(* Schneider Machine Expert - Basic project Water_Heater, file version 1.8.0.0 *)
(* ProjectInformations: Name=New project *)

HARDWARE
  Cpu 0: TM221ME16T/G
  EthernetConfiguration: NetworkName=M221, IpAllocationMode=FixedAddress, IpAddress=100.100.100.102, SubnetMask=255.0.0.0
  SerialLineConfiguration: Baud=Baud19200, Parity=ParityEven, DataBits=DataBits8, StopBits=StopBits1, PhysicalMedium=PhysicalMediumRs485, TransmissionMode=TransmissionModeModbusRtu, SlaveId=1, Addressing=SlaveAddressing
  MastTask: UsePeriodScanMode=false, PeriodScan=100
  FastTask: Period=255
  CpuBehavior: StartingMode=StartAsPreviousState, AutoSaveRamOnEeprom=true, WatchdogPeriod=250

SYMBOLS  (address, symbol, comment, settings)
  %M0       HEATER_MIRROR
  %M1       HEATER_AUTO
  %M2       HEATER_MAN
  %S13      SB_FIRSTRUN  "Indicates the first controller cycle in RUN mode"
  %MW1      CONVERTED_TEMP
  %MW2      SETPOINT
  %MW3      SETPOINT_MIN
  %MW4      MODE_REGISTER
  %MW5      HEATER_CONTROL
  %Q0.0     HEATER

POU New POU
  (* SectionNumber=1 *)

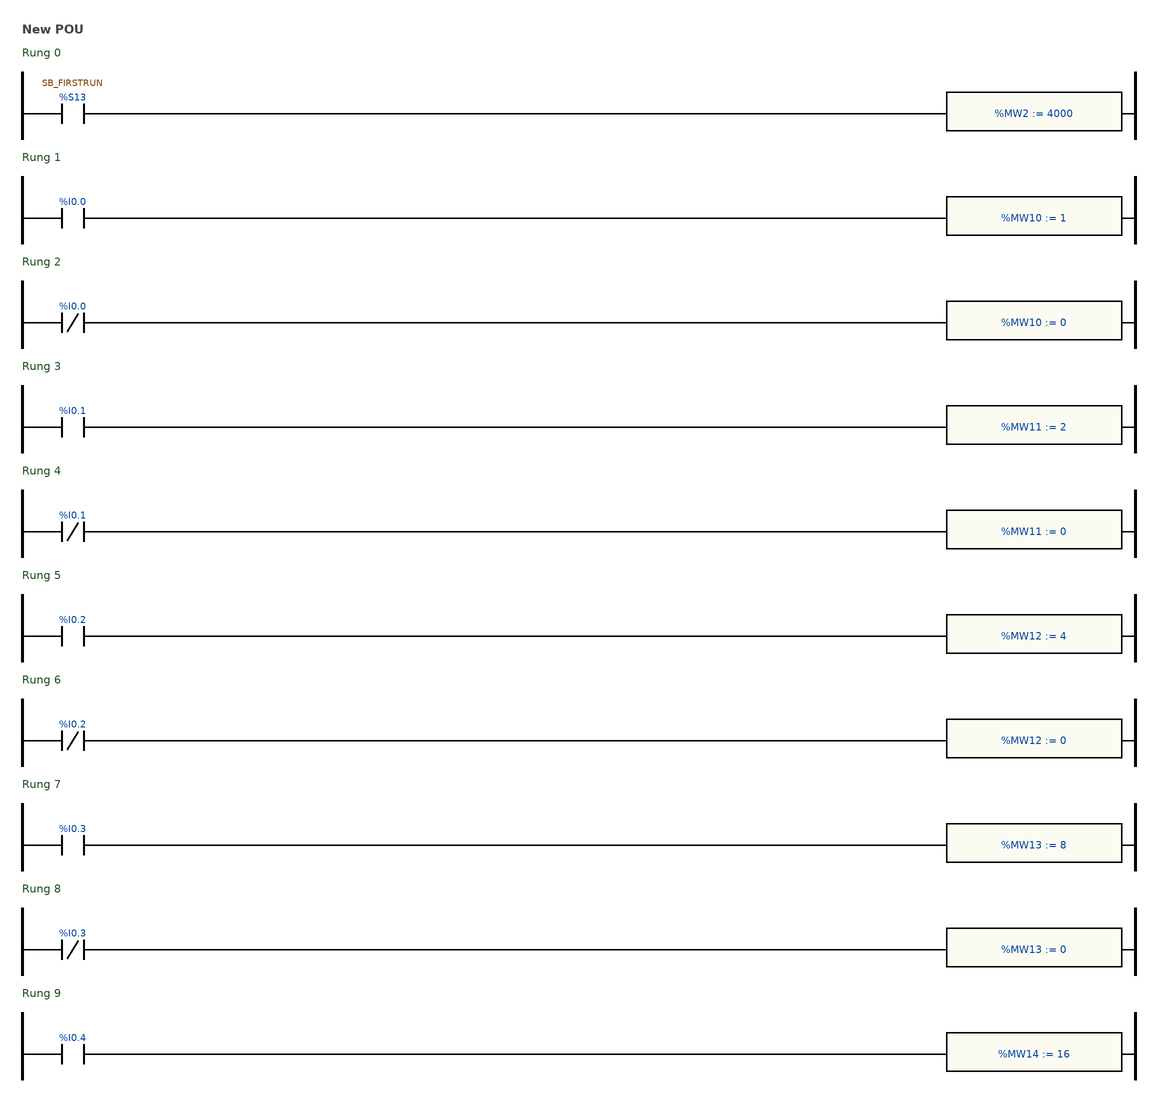

// Rung 0
  LD %S13                 (* SB_FIRSTRUN *)
  [ %MW2 := 4000 ]        (* SETPOINT *)
  // as ST:
  //   IF SB_FIRSTRUN THEN SETPOINT := 4000; END_IF;

// Rung 1
  LD %I0.0
  [ %MW10 := 1 ]
  // as ST:
  //   IF %I0.0 THEN %MW10 := 1; END_IF;

// Rung 2
  LDN %I0.0
  [ %MW10 := 0 ]
  // as ST:
  //   IF NOT %I0.0 THEN %MW10 := 0; END_IF;

// Rung 3
  LD %I0.1
  [ %MW11 := 2 ]
  // as ST:
  //   IF %I0.1 THEN %MW11 := 2; END_IF;

// Rung 4
  LDN %I0.1
  [ %MW11 := 0 ]
  // as ST:
  //   IF NOT %I0.1 THEN %MW11 := 0; END_IF;

// Rung 5
  LD %I0.2
  [ %MW12 := 4 ]
  // as ST:
  //   IF %I0.2 THEN %MW12 := 4; END_IF;

// Rung 6
  LDN %I0.2
  [ %MW12 := 0 ]
  // as ST:
  //   IF NOT %I0.2 THEN %MW12 := 0; END_IF;

// Rung 7
  LD %I0.3
  [ %MW13 := 8 ]
  // as ST:
  //   IF %I0.3 THEN %MW13 := 8; END_IF;

// Rung 8
  LDN %I0.3
  [ %MW13 := 0 ]
  // as ST:
  //   IF NOT %I0.3 THEN %MW13 := 0; END_IF;

// Rung 9
  LD %I0.4
  [ %MW14 := 16 ]
  // as ST:
  //   IF %I0.4 THEN %MW14 := 16; END_IF;

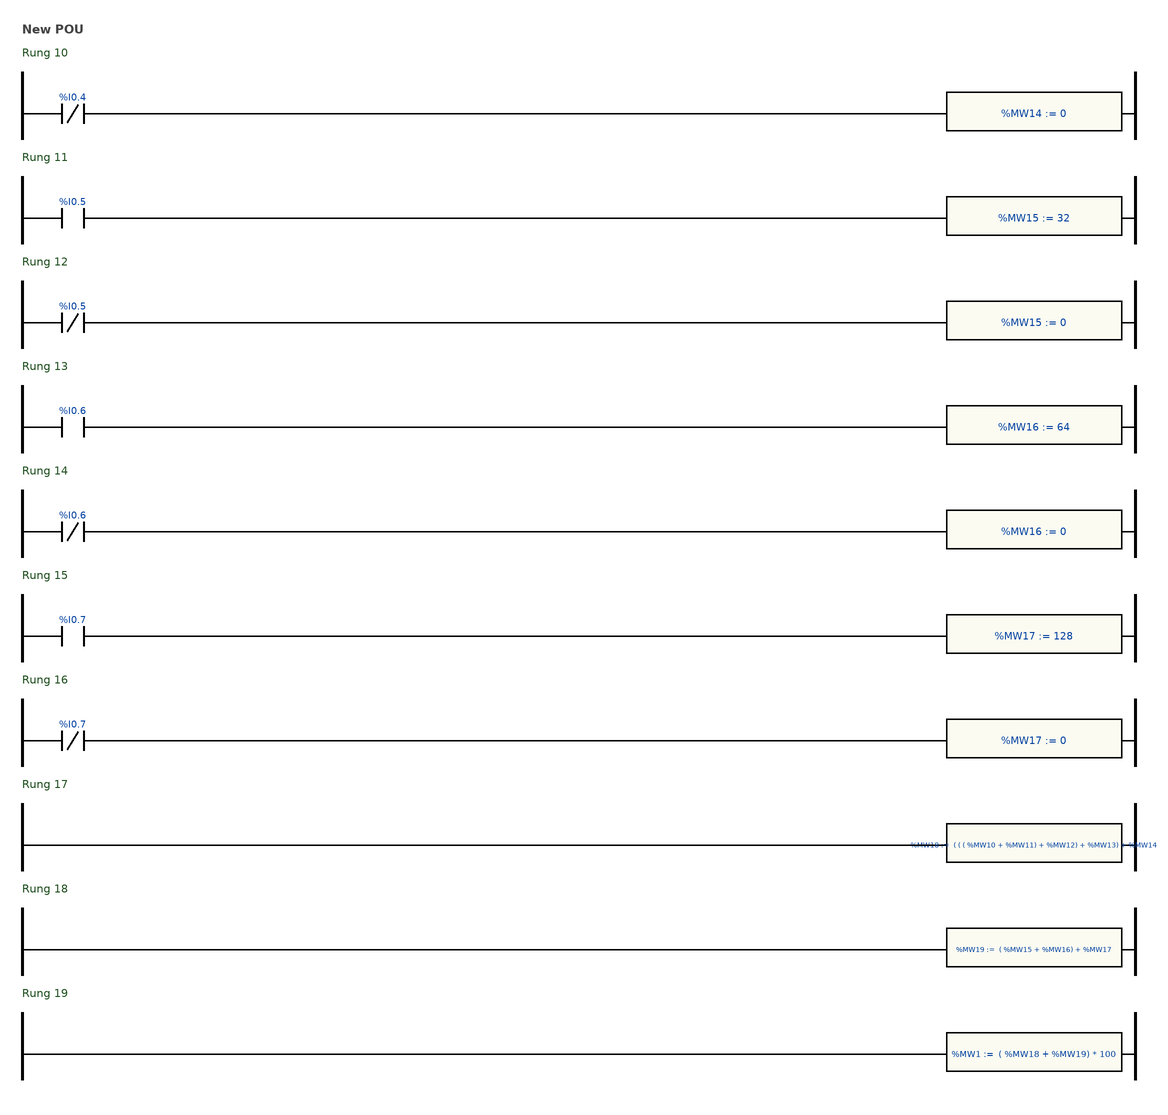

// Rung 10
  LDN %I0.4
  [ %MW14 := 0 ]
  // as ST:
  //   IF NOT %I0.4 THEN %MW14 := 0; END_IF;

// Rung 11
  LD %I0.5
  [ %MW15 := 32 ]
  // as ST:
  //   IF %I0.5 THEN %MW15 := 32; END_IF;

// Rung 12
  LDN %I0.5
  [ %MW15 := 0 ]
  // as ST:
  //   IF NOT %I0.5 THEN %MW15 := 0; END_IF;

// Rung 13
  LD %I0.6
  [ %MW16 := 64 ]
  // as ST:
  //   IF %I0.6 THEN %MW16 := 64; END_IF;

// Rung 14
  LDN %I0.6
  [ %MW16 := 0 ]
  // as ST:
  //   IF NOT %I0.6 THEN %MW16 := 0; END_IF;

// Rung 15
  LD %I0.7
  [ %MW17 := 128 ]
  // as ST:
  //   IF %I0.7 THEN %MW17 := 128; END_IF;

// Rung 16
  LDN %I0.7
  [ %MW17 := 0 ]
  // as ST:
  //   IF NOT %I0.7 THEN %MW17 := 0; END_IF;

// Rung 17
  LD 1
  [%MW18 := ( ( ( %MW10 + %MW11) + %MW12) + %MW13) + %MW14]
  // as ST:
  //   %MW18 :=  ( ( ( %MW10 + %MW11) + %MW12) + %MW13) + %MW14;

// Rung 18
  LD 1
  [%MW19 := ( %MW15 + %MW16) + %MW17]
  // as ST:
  //   %MW19 :=  ( %MW15 + %MW16) + %MW17;

// Rung 19
  LD 1
  [%MW1 := ( %MW18 + %MW19) * 100](* CONVERTED_TEMP *)
  // as ST:
  //   CONVERTED_TEMP :=  ( %MW18 + %MW19) * 100;

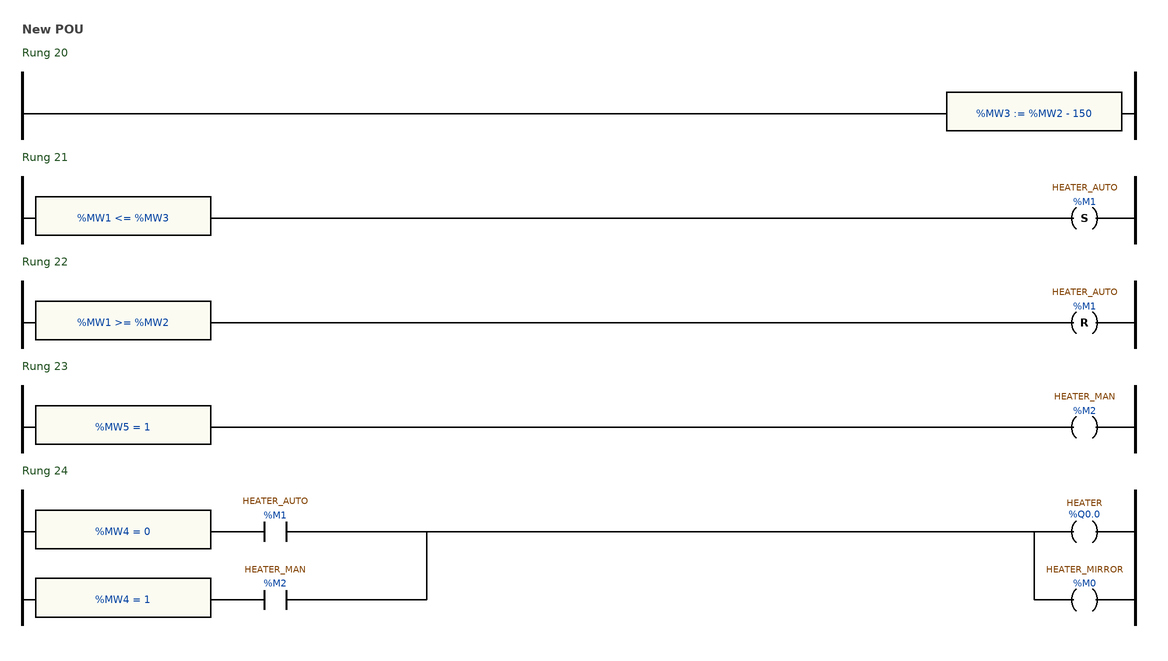

// Rung 20
  LD 1
  [ %MW3 := %MW2 - 150 ]  (* SETPOINT_MIN, SETPOINT *)
  // as ST:
  //   SETPOINT_MIN := SETPOINT - 150;

// Rung 21
  LD [ %MW1 <= %MW3 ]     (* CONVERTED_TEMP, SETPOINT_MIN *)
  S %M1                   (* HEATER_AUTO *)
  // as ST:
  //   IF CONVERTED_TEMP <= SETPOINT_MIN THEN HEATER_AUTO := TRUE; END_IF;

// Rung 22
  LD [ %MW1 >= %MW2 ]     (* CONVERTED_TEMP, SETPOINT *)
  R %M1                   (* HEATER_AUTO *)
  // as ST:
  //   IF CONVERTED_TEMP >= SETPOINT THEN HEATER_AUTO := FALSE; END_IF;

// Rung 23
  LD [ %MW5 = 1 ]         (* HEATER_CONTROL *)
  ST %M2                  (* HEATER_MAN *)
  // as ST:
  //   HEATER_MAN := HEATER_CONTROL = 1;

// Rung 24
  LD [ %MW4 = 0 ]         (* MODE_REGISTER *)
  AND %M1                 (* HEATER_AUTO *)
  OR( [ %MW4 = 1 ]        (* MODE_REGISTER *)
  AND %M2                 (* HEATER_MAN *)
  )
  ST %Q0.0                (* HEATER *)
  ST %M0                  (* HEATER_MIRROR *)
  // as ST:
  //   HEATER := MODE_REGISTER = 0 AND HEATER_AUTO OR MODE_REGISTER = 1 AND HEATER_MAN;
  //   HEATER_MIRROR := MODE_REGISTER = 0 AND HEATER_AUTO OR MODE_REGISTER = 1 AND HEATER_MAN;
